// LS Electric XG5000 project: SV_ CT FRT SEMI MODULE LINE
// PLC LSPLC
// module base 0 slot 0: 입출력 모듈:XBM-DN32H (DC 24V입력/TR 출력, 32점)

PROGRAM VISION (task: 스캔 프로그램)

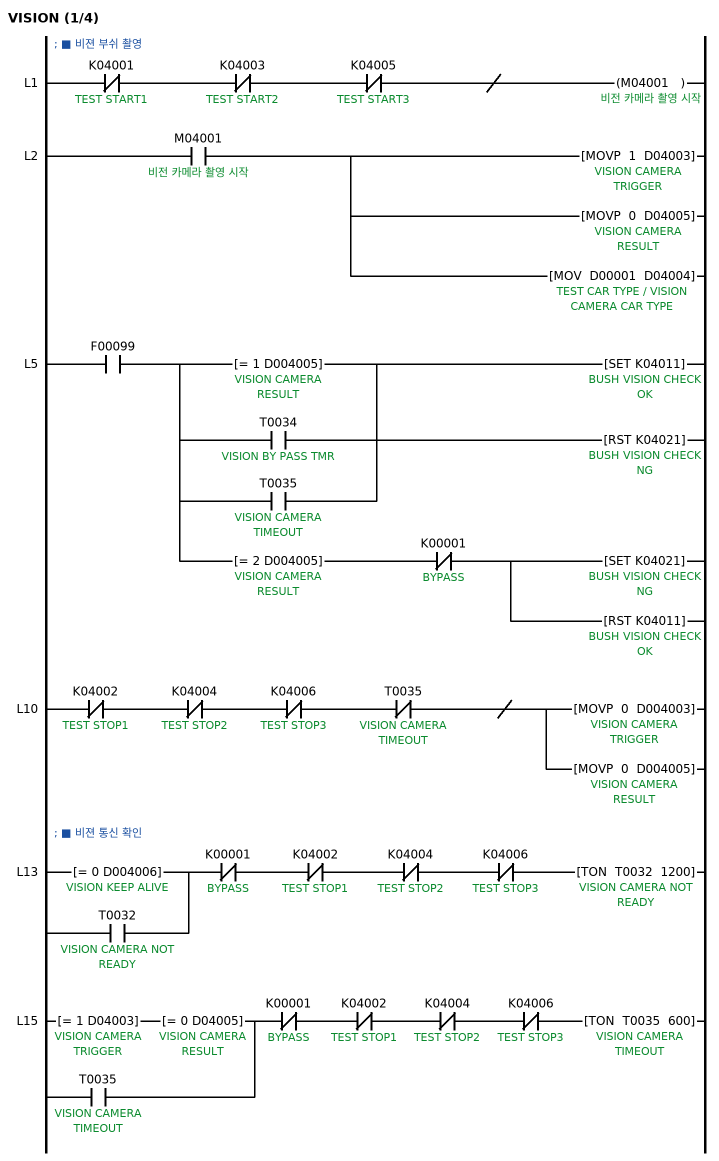
//  ■ 비젼 부쉬 촬영
; L1
LOAD NOT  K04001	// TEST START1
AND NOT   K04003	// TEST START2
AND NOT   K04005	// TEST START3
NOT
OUT       M04001	// 비전 카메라 촬영 시작
; L2
LOAD      M04001	// 비전 카메라 촬영 시작
MOVP      1 D04003	// VISION CAMERA TRIGGER
MOVP      0 D04005	// VISION CAMERA RESULT
MOV       D00001 D04004	// TEST CAR TYPE / VISION CAMERA CAR TYPE
; L5
LOAD      F00099
MPUSH
LOAD=     1 D004005	// VISION CAMERA RESULT
OR        T0034	// VISION BY PASS TMR
OR        T0035	// VISION CAMERA TIMEOUT
AND LOAD
SET       K04011	// BUSH VISION CHECK OK
RST       K04021	// BUSH VISION CHECK NG
MPOP
AND=      2 D004005	// VISION CAMERA RESULT
AND NOT   K00001	// BYPASS
SET       K04021	// BUSH VISION CHECK NG
RST       K04011	// BUSH VISION CHECK OK
; L10
LOAD NOT  K04002	// TEST STOP1
AND NOT   K04004	// TEST STOP2
AND NOT   K04006	// TEST STOP3
AND NOT   T0035	// VISION CAMERA TIMEOUT
NOT
MOVP      0 D004003	// VISION CAMERA TRIGGER
MOVP      0 D004005	// VISION CAMERA RESULT
//  ■ 비젼 통신 확인
; L13
LOAD=     0 D004006	// VISION KEEP ALIVE
OR        T0032	// VISION CAMERA NOT READY
AND NOT   K00001	// BYPASS
AND NOT   K04002	// TEST STOP1
AND NOT   K04004	// TEST STOP2
AND NOT   K04006	// TEST STOP3
TON       T0032 1200	// VISION CAMERA NOT READY
; L15
LOAD=     1 D04003	// VISION CAMERA TRIGGER
AND=      0 D04005	// VISION CAMERA RESULT
OR        T0035	// VISION CAMERA TIMEOUT
AND NOT   K00001	// BYPASS
AND NOT   K04002	// TEST STOP1
AND NOT   K04004	// TEST STOP2
AND NOT   K04006	// TEST STOP3
TON       T0035 600	// VISION CAMERA TIMEOUT

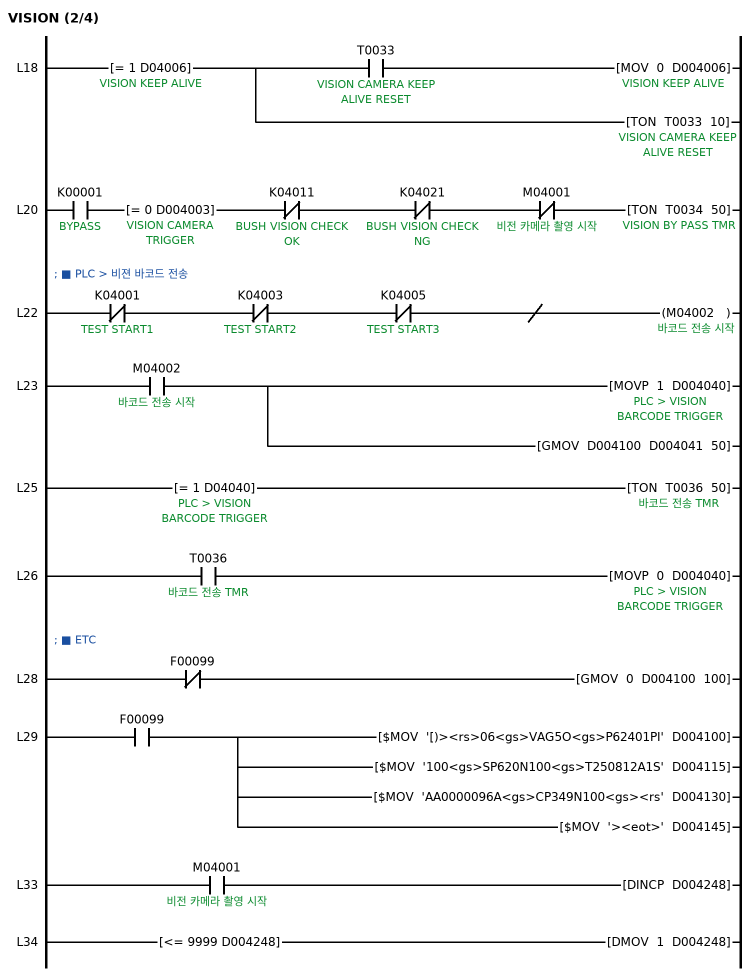
; L18
LOAD=     1 D04006	// VISION KEEP ALIVE
MPUSH
AND       T0033	// VISION CAMERA KEEP ALIVE RESET
MOV       0 D004006	// VISION KEEP ALIVE
MPOP
TON       T0033 10	// VISION CAMERA KEEP ALIVE RESET
; L20
LOAD      K00001	// BYPASS
AND=      0 D004003	// VISION CAMERA TRIGGER
AND NOT   K04011	// BUSH VISION CHECK OK
AND NOT   K04021	// BUSH VISION CHECK NG
AND NOT   M04001	// 비전 카메라 촬영 시작
TON       T0034 50	// VISION BY PASS TMR
//  ■ PLC > 비젼 바코드 전송
; L22
LOAD NOT  K04001	// TEST START1
AND NOT   K04003	// TEST START2
AND NOT   K04005	// TEST START3
NOT
OUT       M04002	// 바코드 전송 시작
; L23
LOAD      M04002	// 바코드 전송 시작
MOVP      1 D004040	// PLC > VISION BARCODE TRIGGER
GMOV      D004100 D004041 50
; L25
LOAD=     1 D04040	// PLC > VISION BARCODE TRIGGER
TON       T0036 50	// 바코드 전송 TMR 
; L26
LOAD      T0036	// 바코드 전송 TMR 
MOVP      0 D004040	// PLC > VISION BARCODE TRIGGER
//  ■ ETC
; L28
LOAD NOT  F00099
GMOV      0 D004100 100
; L29
LOAD      F00099
$MOV      '[)><rs>06<gs>VAG5O<gs>P62401PI' D004100
$MOV      '100<gs>SP620N100<gs>T250812A1S' D004115
$MOV      'AA0000096A<gs>CP349N100<gs><rs' D004130
$MOV      '><eot>' D004145
; L33
LOAD      M04001	// 비전 카메라 촬영 시작
DINCP     D004248
; L34
LOAD<=    9999 D004248
DMOV      1 D004248

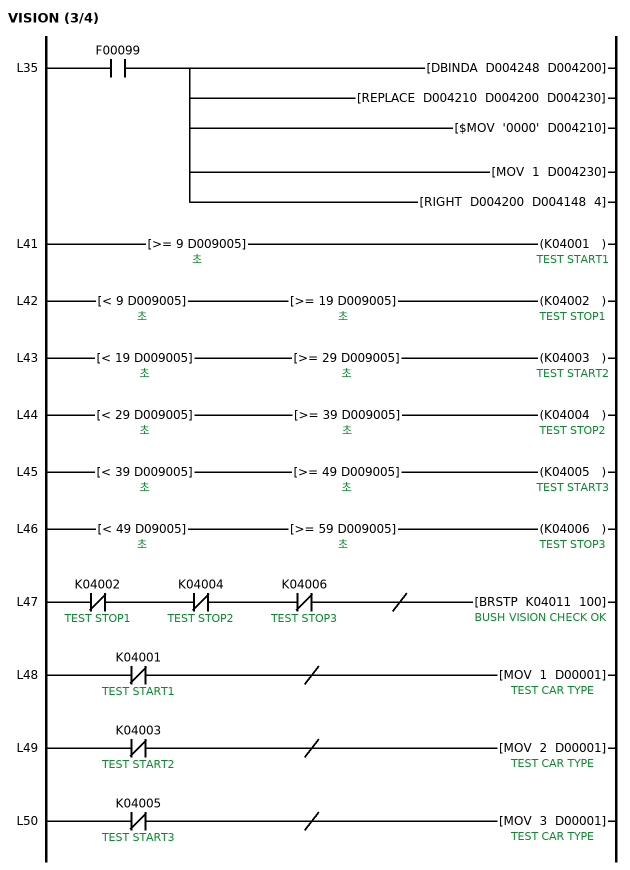
; L35
LOAD      F00099
DBINDA    D004248 D004200
REPLACE   D004210 D004200 D004230
$MOV      '0000' D004210
MOV       1 D004230
RIGHT     D004200 D004148 4
; L41
LOAD>=    9 D009005	// 초
OUT       K04001	// TEST START1
; L42
LOAD<     9 D009005	// 초
AND>=     19 D009005	// 초
OUT       K04002	// TEST STOP1
; L43
LOAD<     19 D009005	// 초
AND>=     29 D009005	// 초
OUT       K04003	// TEST START2
; L44
LOAD<     29 D009005	// 초
AND>=     39 D009005	// 초
OUT       K04004	// TEST STOP2
; L45
LOAD<     39 D009005	// 초
AND>=     49 D009005	// 초
OUT       K04005	// TEST START3
; L46
LOAD<     49 D09005	// 초
AND>=     59 D009005	// 초
OUT       K04006	// TEST STOP3
; L47
LOAD NOT  K04002	// TEST STOP1
AND NOT   K04004	// TEST STOP2
AND NOT   K04006	// TEST STOP3
NOT
BRSTP     K04011 100	// BUSH VISION CHECK OK
; L48
LOAD NOT  K04001	// TEST START1
NOT
MOV       1 D00001	// TEST CAR TYPE
; L49
LOAD NOT  K04003	// TEST START2
NOT
MOV       2 D00001	// TEST CAR TYPE
; L50
LOAD NOT  K04005	// TEST START3
NOT
MOV       3 D00001	// TEST CAR TYPE

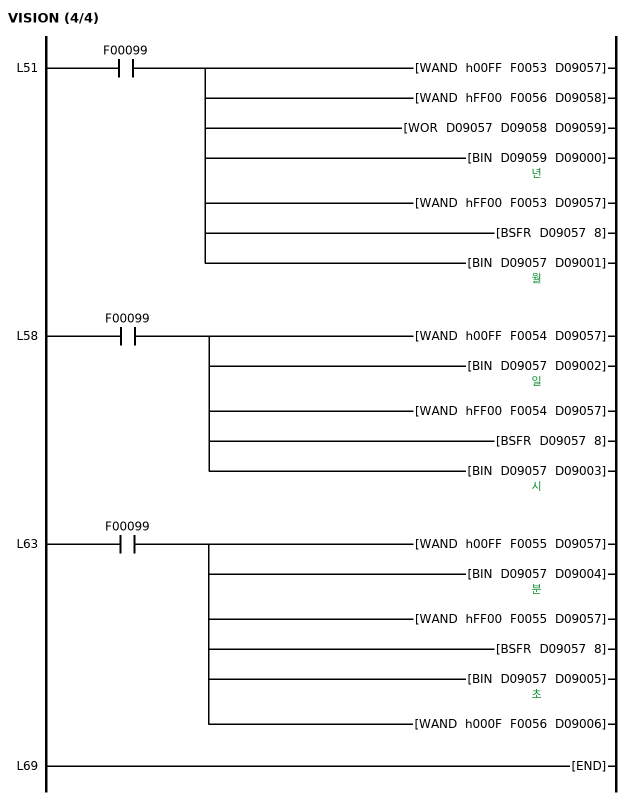
; L51
LOAD      F00099
WAND      h00FF F0053 D09057
WAND      hFF00 F0056 D09058
WOR       D09057 D09058 D09059
BIN       D09059 D09000	// 년
WAND      hFF00 F0053 D09057
BSFR      D09057 8
BIN       D09057 D09001	// 월
; L58
LOAD      F00099
WAND      h00FF F0054 D09057
BIN       D09057 D09002	// 일
WAND      hFF00 F0054 D09057
BSFR      D09057 8
BIN       D09057 D09003	// 시
; L63
LOAD      F00099
WAND      h00FF F0055 D09057
BIN       D09057 D09004	// 분
WAND      hFF00 F0055 D09057
BSFR      D09057 8
BIN       D09057 D09005	// 초
WAND      h000F F0056 D09006
; L69
END

VARIABLES AND COMMENTS (devices not used above)
D06000	WORD	OCR Trig
D06001	WORD	OCR Model
D06006	WORD	Vision Ready
K00591	BIT	CAR TYPE TMA 2WD
K00592	BIT	CAR TYPE TMA 4WD
K00593	BIT	CAR TYPE ON 2WD
K00594	BIT	CAR TYPE ON 4WD
T0001	BIT/WORD	Welding Bead Trig ON
T0002	BIT/WORD	Trig OFF
P00020	BIT	OCR Trig
P00021	BIT	Visin Trig
T0000	BIT/WORD	first time ON
T0010	BIT/WORD	OCR Trig time ready
M00020	BIT	OCR finish
T0020	BIT/WORD	Camera trig time
T0030	BIT/WORD	Camera finish time 
M00010	BIT	Camer finish
T0005	BIT/WORD	Reset time
D06002	WORD	OCR result
D06005	WORD	camera result
D06003	WORD	camera Trig
D06004	WORD	Camera Model